FUNCTION_BLOCK FB_SaMElementManual EXTENDS FB_SaMElement
VAR
END_VAR

METHOD FB_init : BOOL
VAR_INPUT
	bInitRetains : BOOL; // if TRUE, the retain variables are initialized (warm start / cold start)
	bInCopyCode : BOOL;  // if TRUE, the instance afterwards gets moved into the copy code (online change)
END_VAR
THIS^.SetText (eLocation := E_BaseLocation.pl, wsDescription := "Ręczny");
THIS^.SetText (eLocation := E_BaseLocation.en, wsDescription := "Manual");
THIS^.SetText (eLocation := E_BaseLocation.de, wsDescription := "Handbuch");
THIS^.SetName (stName := THIS^.GetTexts ());
END_METHOD

END_FUNCTION_BLOCK

(* stored: Version 1.1.0.1
   POU FB_SaMElementManual: Id {54e27e12-3d3f-0f17-3788-9da4dcb3548e}, SpecialFunc None
   Method FB_init: Id {b15ce8cd-29f9-0eec-3c14-382a89447901} *)
